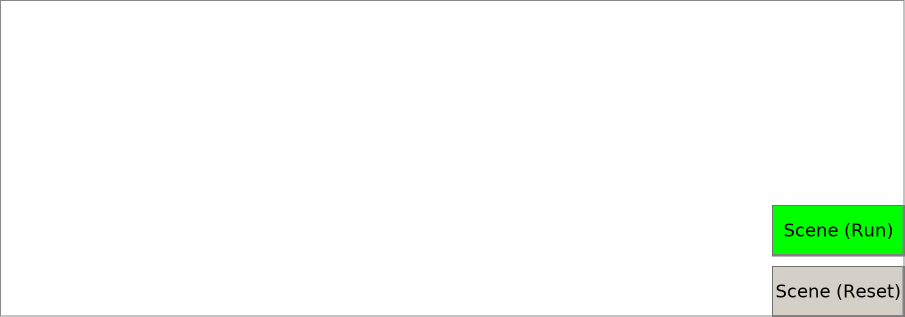
VISUALIZATION Visualization  // 905x317
    Button (772,205 133x51), "Scene (Run)"
        toggle xSystemPower
    Button (772,266 133x51), "Scene (Reset)"
        tap xSystemReset
END_VISUALIZATION

(* stored: Version 1.1.0.1
   Visu Visualization: Id {a0ed1e60-ffdd-493f-977a-e065fc0f75d0} *)
